(* IEC 61131-3 sources: repolevel_ST_code_completion/output/0127完整版本_带planner/repoeval_traffic_light/readful_result_history, 4 files *)

(* ---- F_SecondsToTime_0.st ---- *)
FUNCTION F_SecondsToTime : TIME
VAR_INPUT
	dwSeconds	:	DWORD;		//输入的秒数
END_VAR
F_SecondsToTime := DWORD_TO_TIME(dwSeconds * 1000);
RETURN;
END_FUNCTION

(* ---- F_TimeToSeconds_0.st ---- *)
FUNCTION F_TimeToSeconds : DWORD
VAR_INPUT
	tTime	:	TIME;		//输入的时间
END_VAR
F_TimeToSeconds := DINT_TO_DWORD(TRUNC(TIME_TO_DWORD(tTime) / 1000.0));
RETURN;
END_FUNCTION

(* ---- FB_CountdownTimer_0.st ---- *)
FUNCTION_BLOCK FB_CountdownTimer
VAR_INPUT
	tElapsedTime	:	TIME;		//已经过的时间（定时器的ET）
	tTotalTime		:	TIME;		//总时间（定时器的PT）
END_VAR
VAR_OUTPUT
	nRemainingSeconds	:	UINT;	//剩余秒数
END_VAR
VAR
	nTotalSeconds		:	UINT;	//总秒数
	nElapsedSeconds		:	UINT;	//已过秒数
END_VAR

// 将TIME转换为秒
nTotalSeconds := UINT_TO_UINT(DWORD_TO_UINT(TIME_TO_DWORD(tTotalTime) / 1000));
nElapsedSeconds := UINT_TO_UINT(DWORD_TO_UINT(TIME_TO_DWORD(tElapsedTime) / 1000));

// 检查是否已经过了总时间
IF tElapsedTime >= tTotalTime THEN
	nRemainingSeconds := 0;
ELSE
	// 计算剩余秒数
	nRemainingSeconds := nTotalSeconds - nElapsedSeconds;
END_IF;
END_FUNCTION_BLOCK

(* ---- FB_CountdownTimer_1.st ---- *)
FUNCTION_BLOCK FB_CountdownTimer
VAR_INPUT
	tElapsedTime	:	TIME;		//已经过的时间（定时器的ET）
	tTotalTime		:	TIME;		//总时间（定时器的PT）
END_VAR
VAR_OUTPUT
	nRemainingSeconds	:	UINT;	//剩余秒数
END_VAR
VAR
	nTotalSeconds		:	UINT;	//总秒数
	nElapsedSeconds		:	UINT;	//已过秒数
END_VAR

// 将TIME转换为秒
nTotalSeconds := TO_UINT(TIME_TO_DWORD(tTotalTime) / 1000);
nElapsedSeconds := TO_UINT(TIME_TO_DWORD(tElapsedTime) / 1000);

// 检查是否已经过了总时间
IF tElapsedTime >= tTotalTime THEN
	nRemainingSeconds := 0;
ELSE
	// 计算剩余秒数
	nRemainingSeconds := nTotalSeconds - nElapsedSeconds;
END_IF;
END_FUNCTION_BLOCK
